PROGRAM MAIN
VAR
	fbMainloop	: fb_Conveyor;
END_VAR

fbMainloop();

//Output to Virtual Machine
DataExchange.nAcceleration := fbMainloop.nAcceleration;
DataExchange.nDeceleration := fbMainloop.nDeceleration;
DataExchange.nDirection := fbMainloop.nDirection;
DataExchange.nVelocity := fbMainloop.nVelocity;
DataExchange.bAxis := fbMainloop.bAxis;
DataExchange.bHalt := fbMainloop.bHalt;


//Input from Virtual Machine
fbMainloop.bS1 := DataExchange.bS1;
fbMainloop.bS2 := DataExchange.bS2;
fbMainloop.bS3 := DataExchange.bS3;
fbMainloop.bInVelocity := DataExchange.bInVelocity;

END_PROGRAM

(* stored: Version 1.1.0.1, ProductVersion 3.1.4024.12
   POU MAIN: Id {75e5defc-e010-45e4-a563-69e838af7978}, SpecialFunc None *)
